FUNCTION_BLOCK FB_UniversalVFDModbus_Ex EXTENDS FB_UniversalVFDModbus

SUPER^();

METHOD Convert : BOOL
VAR_INPUT
	iRegionNo	:	INT;
	pReadData	:	POINTER TO word;
END_VAR
CASE iRegionNo OF
	0:
		IF pReadData[0] = 10 THEN
			eVfdStatus := VFD_STATUS_READY_TO_RUN;
		END_IF
END_CASE
END_METHOD

END_FUNCTION_BLOCK

(* stored: Version 1.1.0.1, ProductVersion 3.1.4024.12
   POU FB_UniversalVFDModbus_Ex: Id {525cf8e8-ff46-40d7-a282-18fc349596ed}, SpecialFunc None
   Method Convert: Id {8473276c-a2e5-4241-a5e0-333391def56e} *)
